{attribute 'linkalways'} 
{attribute 'no_explicit_call' := 'This FB is a CLASS and must be accessed using methods or properties'}
{attribute 'enable_dynamic_creation'}
FUNCTION_BLOCK Node_F_VN_InsertIntoContainer_TcVnVector2_USINT EXTENDS VisionNode
VAR
    aElement : _TcVnVector2_USINT;
    ipContainer : _ITcVnContainer;
    nIndex : _ULINT(0);
    hrPrev : _HRESULT(S_OK);
    hresult : _HRESULT(S_OK);
END_VAR

METHOD PUBLIC  Clone : I_Node
VAR
	pNode : POINTER TO Node_F_VN_InsertIntoContainer_TcVnVector2_USINT;
END_VAR
pNode := __NEW(Node_F_VN_InsertIntoContainer_TcVnVector2_USINT);
Clone := pNode^;
END_METHOD

METHOD FB_init : BOOL
VAR_INPUT
	bInitRetains : BOOL; // if TRUE, the retain variables are initialized (warm start / cold start)
	bInCopyCode : BOOL;  // if TRUE, the instance afterwards gets moved into the copy code (online change)
END_VAR
AddInput('aElement', aElement);
AddInput('ipContainer', ipContainer);
AddInput('nIndex', nIndex);
AddInput('hrPrev', hrPrev);
AddOutput('ipContainer', ipContainer);
AddOutput('hresult',hresult);
END_METHOD

METHOD PROTECTED OnExecute : HRESULT
hresult.Value := F_VN_InsertIntoContainer_TcVnVector2_USINT(
    aElement := aElement.Value,
    ipContainer := ipContainer.Value,
    nIndex := nIndex.Value,
    hrPrev:= hrPrev.Value);
END_METHOD

METHOD PUBLIC PreExecutionCheck
VAR_INPUT
	Check : I_PreExecutionChecks;
END_VAR
Check.IsTrue(ipContainer.IsValid, 'ipContainer must be a valid container');
END_METHOD

END_FUNCTION_BLOCK

(* stored: Version 1.1.0.1, ProductVersion 3.1.4024.13
   POU Node_F_VN_InsertIntoContainer_TcVnVector2_USINT: Id {c6b75654-7ce7-465b-98a8-80b6cc247695}, SpecialFunc None
   Folder Constructor: Id {9a60c22a-f295-48ee-b178-4e16fd000704}
   Method Clone: Id {98dc1994-767f-459f-94f7-7761caee84c3}
   Method FB_init: Id {2c1ddc51-a4b4-4d70-ae94-1b7ced652abb}
   Method OnExecute: Id {d671307d-bf4d-4b6a-b9f8-76475c1ffcd8}
   Method PreExecutionCheck: Id {616e8a1b-ca53-4a10-b5b5-fab1fd34d3a8} *)
